// LS Electric XG5000 project: project D
// PLC NewPLC
// module base 0 slot 0: 입출력 모듈:XBC-DR32H (DC 24V 입력, 릴레이 출력 32점)

PROGRAM NewProgram (task: 스캔 프로그램)

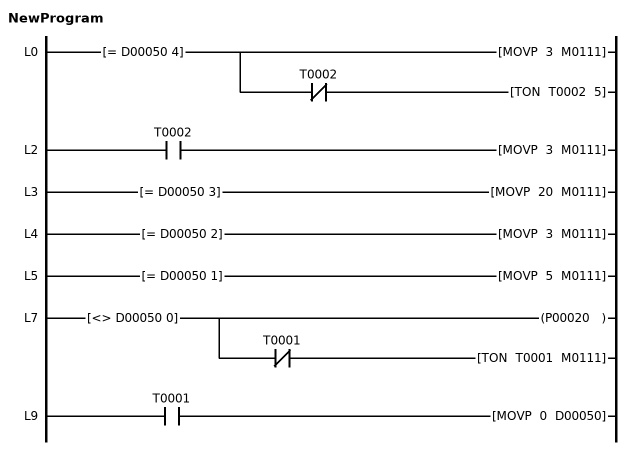
; L0
LOAD=     D00050 4
MOVP      3 M0111
AND NOT   T0002
TON       T0002 5
; L2
LOAD      T0002
MOVP      3 M0111
; L3
LOAD=     D00050 3
MOVP      20 M0111
; L4
LOAD=     D00050 2
MOVP      3 M0111
; L5
LOAD=     D00050 1
MOVP      5 M0111
; L7
LOAD<>    D00050 0
OUT       P00020
AND NOT   T0001
TON       T0001 M0111
; L9
LOAD      T0001
MOVP      0 D00050